// TIA Portal V19 export
VAR_GLOBAL   // PLC tag table "PTRK"
END_VAR
VAR_GLOBAL CONSTANT   // user constants
   PTRK_A0202_ITEMS : Int := 15;
   PTRK_A0202_EXIT_TOCHECK_ITEMS : Int := 10;
   PTRK_A0301_ITEMS : Int := 20;
END_VAR
